RESOURCE_TYPE {name} (* Resource Type *)
  (* Standard: 61499-2 *)
  (* Version 0.0, {date}, {author}, NetAllied *)
END_RESOURCE_TYPE
